# B&R Automation Studio project baseProject (part 2)

#### Main.st
```iecst
PROGRAM _INIT

	//Enable FBs and set parameters
	MpSequenceCore_0.Enable := TRUE;
	MpSequenceCore_0.Import := TRUE;
	MpSequenceCore_0.Mode := mpSEQUENCE_MODE_SINGLE_CYCLE;
	ParametersCore.Sequence := 'CoffeeSequence.xml';

	Timer.AxisLeft.PT := T#03s;
	Timer.AxisRight.PT := T#03s;
	Timer.Coffee.PT := T#03s;
	Timer.ExecuteWait.PT := T#03s;
	Timer.Start.PT := T#500ms;
	Timer.Stop.PT := T#01s;
	Timer.TakeOutCup.PT := T#01s;
	Timer.Wait.PT := T#03s;
	Timer.StopButton.PT := T#02s;
	Timer.CoffeeWait.PT := T#01s;

END_PROGRAM
PROGRAM _CYCLIC

	//Set FB parameters
	MpSequenceCore_0.MpLink := ADR(gSequenceCore);
	MpSequenceCore_0.Parameters := ADR(ParametersCore);

	IF MpSequenceCore_0.CommandDone AND MpSequenceCore_0.Import THEN
		MpSequenceCore_0.Import := FALSE;
	END_IF

	//Start if Start-Button is pressed
	IF SequenceStart AND MpSequenceCore_0.Info.ReadyToStart THEN
		MpSequenceCore_0.Start := TRUE;
		EditSequence := FALSE;
		MpSequenceCore_0.ErrorReset := FALSE;
	ELSE

		MpSequenceCore_0.Start := FALSE;
		CmdSeq.Start.MovementState := mpSEQUENCE_MOVEMENT_IDLE;
		CmdSeq.AxisLeft.MovementState := mpSEQUENCE_MOVEMENT_IDLE;
		CmdSeq.AxisRight.MovementState := mpSEQUENCE_MOVEMENT_IDLE;
		CmdSeq.Coffee.MovementState := mpSEQUENCE_MOVEMENT_IDLE;
		CmdSeq.End.MovementState := mpSEQUENCE_MOVEMENT_IDLE;
		CmdSeq.TakeOutCup.MovementState := mpSEQUENCE_MOVEMENT_IDLE;
		CmdSeq.Wait.MovementState := mpSEQUENCE_MOVEMENT_IDLE;
		Timer.AxisLeft.IN := FALSE;
		Timer.AxisRight.IN := FALSE;
		Timer.Coffee.IN := FALSE;
		Timer.ExecuteWait.IN := FALSE;
		Timer.Start.IN := FALSE;
		Timer.Stop.IN := FALSE;
		Timer.TakeOutCup.IN := FALSE;
		Timer.Wait.IN := FALSE;
		Timer.StopButton.IN := TRUE;

		Transform := '[{"select":"#g83","duration":1000,"translate":[3.497,-208.81101],"display":true}
		,{"select":"#rect999-9-2","duration":1000,"display":false}
		,{"select":"#rect999-1","duration":1000,"display":false}
		,{"select":"#path49","duration":2000,"fill":7}
		,{"select":"#path39","duration":2000,"fill":0}
		,{"select":"#path41","duration":2000,"fill":2}
		,{"select":"#path3","duration":2000,"fill":3}
		,{"select":"#gLamp1","duration":2000,"fill":7}
		,{"select":"#gLamp2","duration":2000,"fill":7}
		,{"select":"#gLamp3","duration":2000,"fill":7}
		,{"select":"#gLamp4","duration":2000,"fill":7}
		,{"select":"#gLamp5","duration":2000,"fill":7}
		,{"select":"#gLamp6","duration":2000,"fill":7}]';

		IF Timer.StopButton.Q THEN
			Timer.StopButton.IN := FALSE;
		END_IF

		EditSequence := TRUE;

	END_IF

	(****************************************************************START*********************************************************************)
	IF CmdSeq.Start.Start THEN

		CmdSeq.Start.MovementState := mpSEQUENCE_MOVEMENT_ACTIVE;
		Timer.Start.IN := TRUE;
		Transform := '[{"select":"#g83","duration":500,"display":true}]';
		IF Timer.Start.Q THEN
			Timer.Start.IN := FALSE;
			CmdSeq.Start.MovementState := mpSEQUENCE_MOVEMENT_DONE;
		END_IF

	ELSE
		CmdSeq.Start.MovementState := mpSEQUENCE_MOVEMENT_IDLE;
	END_IF

	(****************************************************************AXIS LEFT*********************************************************************)
	IF CmdSeq.AxisLeft.Start THEN

		CmdSeq.AxisLeft.MovementState := mpSEQUENCE_MOVEMENT_ACTIVE;
		Timer.AxisLeft.IN := TRUE;
		Transform := '[{"select":"#g83","duration":3000,"translate":[440,-208.81101]},{"select":"#gLamp1","duration":2000,"fill":8},{"select":"#gLamp4","duration":2000,"fill":8}]';
		IF Timer.AxisLeft.Q THEN
			Timer.AxisLeft.IN := FALSE;
			CmdSeq.AxisLeft.MovementState := mpSEQUENCE_MOVEMENT_DONE;
		END_IF
	ELSE
		CmdSeq.AxisLeft.MovementState := mpSEQUENCE_MOVEMENT_IDLE;
	END_IF

	(****************************************************************AXIS RIGHT*********************************************************************)
	IF CmdSeq.AxisRight.Start THEN

		CmdSeq.AxisRight.MovementState := mpSEQUENCE_MOVEMENT_ACTIVE;
		Timer.AxisRight.IN := TRUE;
		Transform := '[{"select":"#g83","duration":3000,"translate":[560,-208.81101]},{"select":"#gLamp3","duration":2000,"fill":10},{"select":"#gLamp6","duration":2000,"fill":10}]';
		IF Timer.AxisRight.Q THEN
			Timer.AxisRight.IN := FALSE;
			CmdSeq.AxisRight.MovementState := mpSEQUENCE_MOVEMENT_DONE;
		END_IF
	ELSE
		CmdSeq.AxisRight.MovementState := mpSEQUENCE_MOVEMENT_IDLE;
	END_IF

	(****************************************************************COFFEE*********************************************************************)
	IF CmdSeq.Coffee.Start THEN

		CmdSeq.Coffee.MovementState := mpSEQUENCE_MOVEMENT_ACTIVE;
		Timer.Coffee.IN := TRUE;
		Transform :='[{"select":"#path39","duration":2000,"fill":7}
		,{"select":"#path41","duration":2000,"fill":7}
		,{"select":"#path3","duration":2000,"fill":7}
		,{"select":"#gLamp2","duration":2000,"fill":9},
		{"select":"#gLamp5","duration":2000,"fill":9}]';
		IF Timer.Coffee.Q THEN

			Timer.ExecuteWait.IN := TRUE;

			Transform := '[{"select":"#rect999-9-2","duration":2000,"display":true,"fill":1}
			,{"select":"#rect999-1","duration":2000,"display":true,"fill":1}
			,{"select":"#path49","duration":2000,"fill":0}
			,{"select":"#path39","duration":2000,"fill":0}
			,{"select":"#path41","duration":2000,"fill":2}
			,{"select":"#path3","duration":2000,"fill":3}]';
			IF Timer.ExecuteWait.Q THEN

				Timer.CoffeeWait.IN := TRUE;
				Transform := '[{"select":"#rect999-1","duration":1000,"display":false},
				{"select":"#rect999-9-2","duration":1000,"display":false},
				{"select":"#path49","duration":1000,"fill":7}]';
				IF Timer.CoffeeWait.Q THEN
					Timer.CoffeeWait.IN := FALSE;
					Timer.Coffee.IN := FALSE;
					Timer.ExecuteWait.IN := FALSE;
					CmdSeq.Coffee.MovementState := mpSEQUENCE_MOVEMENT_DONE;
				END_IF
			END_IF
		END_IF

	ELSE
		CmdSeq.Coffee.MovementState := mpSEQUENCE_MOVEMENT_IDLE;
	END_IF

	(****************************************************************TAKEOUT*********************************************************************)
	IF CmdSeq.TakeOutCup.Start THEN

		CmdSeq.TakeOutCup.MovementState := mpSEQUENCE_MOVEMENT_ACTIVE;
		Timer.TakeOutCup.IN := TRUE;
		Transform := '[{"select":"#g83","duration":500,"display":false}]';
		IF Timer.TakeOutCup.Q THEN
			Timer.TakeOutCup.IN := FALSE;
			CmdSeq.TakeOutCup.MovementState := mpSEQUENCE_MOVEMENT_DONE;
		END_IF
	ELSE
		CmdSeq.TakeOutCup.MovementState := mpSEQUENCE_MOVEMENT_IDLE;
	END_IF

	(****************************************************************WAIT*********************************************************************)
	IF CmdSeq.Wait.Start THEN
		CmdSeq.Wait.MovementState := mpSEQUENCE_MOVEMENT_ACTIVE;
		Timer.Wait.IN := TRUE;

		IF Timer.Wait.Q THEN
			Timer.Wait.IN := FALSE;
			CmdSeq.Wait.MovementState := mpSEQUENCE_MOVEMENT_DONE;
		END_IF
	ELSE
		CmdSeq.Wait.MovementState := mpSEQUENCE_MOVEMENT_IDLE;
	END_IF

	(****************************************************************STOP*********************************************************************)
	IF CmdSeq.Stop.Start THEN
		CmdSeq.Stop.MovementState := mpSEQUENCE_MOVEMENT_ACTIVE;
		Timer.Stop.IN := TRUE;
		Transform := '[{"select":"#g83","duration":1000,"translate":[3.497,-208.81101]}
		]';

		IF Timer.Stop.Q THEN
			Timer.Stop.IN := FALSE;
			CmdSeq.Stop.MovementState := mpSEQUENCE_MOVEMENT_DONE;
			Transform := '[{"select":"#g83","duration":500,"display":true}]';
			SequenceStart := FALSE;
		END_IF
	ELSE
		CmdSeq.Stop.MovementState := mpSEQUENCE_MOVEMENT_IDLE;
	END_IF

	(****************************************************************ERROR*********************************************************************)
	IF MpSequenceCore_0.Error THEN
		SequenceStart := FALSE;
		MpSequenceCore_0.Import := FALSE;
		MpSequenceCore_0.ErrorReset := gCoffeeMainLogic.cmdClear;
	END_IF

	IF SavePressed THEN
		MpSequenceCore_0.Import := TRUE;
		SavePressed := FALSE;
	END_IF

	//Call FB
	MpSequenceCore_0();
	Timer.AxisLeft();
	Timer.AxisRight();
	Timer.Coffee();
	Timer.Start();
	Timer.Stop();
	Timer.TakeOutCup();
	Timer.Wait();
	Timer.ExecuteWait();
	Timer.StopButton();
	Timer.CoffeeWait();

END_PROGRAM
```

### Program Logical/Infrastructure/CodeBox (IEC) - CodeBox handling

#### Main.st
```iecst
PROGRAM _INIT

	State := WAIT;

END_PROGRAM

PROGRAM _CYCLIC

	//Set FB parameter
	MpCodeBoxCore_0(
	MpLink := ADR(gCodeBoxCore),
	Enable := TRUE,
	ErrorReset := gCoffeeMainLogic.cmdClear);

	CASE State OF
		WAIT:
			CodeBoxTransform := '[{"select":"#gLamp1","duration":200,"fill":7}
			,{"select":"#gLamp2","duration":200,"fill":7}
			,{"select":"#gLamp3","duration":200,"fill":7}
			,{"select":"#gLamp4","duration":200,"fill":7}
			,{"select":"#gLamp5","duration":200,"fill":7}
			,{"select":"#gLamp6","duration":200,"fill":7}]';

			IF gCoffeeMainLogic.PackMLState = 'Idle' THEN
				State := CUP_START_POS;

			END_IF

		CUP_START_POS:
			Cup.StartPosition := TRUE;
			IF Lamp.Green THEN

				CodeBoxTransform := '[{"select":"#gLamp1","duration":1000,"fill":10}
					,{"select":"#gLamp2","duration":1000,"fill":7}
					,{"select":"#gLamp3","duration":1000,"fill":7}
					,{"select":"#gLamp4","duration":1000,"fill":10}
					,{"select":"#gLamp5","duration":1000,"fill":7}
					,{"select":"#gLamp6","duration":1000,"fill":7}]';

			ELSIF Lamp.Red THEN
				CodeBoxTransform := '[{"select":"#gLamp1","duration":1000,"fill":8}
				,{"select":"#gLamp2","duration":1000,"fill":7}
				,{"select":"#gLamp3","duration":1000,"fill":7}
				,{"select":"#gLamp4","duration":1000,"fill":8}
				,{"select":"#gLamp5","duration":1000,"fill":7}
				,{"select":"#gLamp6","duration":1000,"fill":7}]';

			ELSIF Lamp.Yellow THEN
				CodeBoxTransform := '[{"select":"#gLamp1","duration":1000,"fill":9}
				,{"select":"#gLamp2","duration":1000,"fill":7}
				,{"select":"#gLamp3","duration":1000,"fill":7}
				,{"select":"#gLamp4","duration":1000,"fill":9}
				,{"select":"#gLamp5","duration":1000,"fill":7}
				,{"select":"#gLamp6","duration":1000,"fill":7}]';
			ELSE
				CodeBoxTransform := '[{"select":"#gLamp1","duration":1000,"fill":7}
				,{"select":"#gLamp2","duration":1000,"fill":7}
				,{"select":"#gLamp3","duration":1000,"fill":7}
				,{"select":"#gLamp4","duration":1000,"fill":7}
				,{"select":"#gLamp5","duration":1000,"fill":7}
				,{"select":"#gLamp6","duration":1000,"fill":7}]';
			END_IF

			IF gCoffeeMainLogic.PackMLState = 'Execute' THEN
				State := CUP_COFFEE;
				Cup.StartPosition := FALSE;
			END_IF

		CUP_COFFEE:
			Cup.CoffeePosition := TRUE;
			IF gCoffeeMainLogic.PackMLState = 'Completing' THEN
				State := CUP_END_POS;
				Cup.CoffeePosition := FALSE;
			END_IF

			IF Lamp.Green THEN

				CodeBoxTransform := '[{"select":"#gLamp1","duration":1000,"fill":7}
				,{"select":"#gLamp2","duration":1000,"fill":10}
				,{"select":"#gLamp3","duration":1000,"fill":7}
				,{"select":"#gLamp4","duration":1000,"fill":7}
				,{"select":"#gLamp5","duration":1000,"fill":10}
				,{"select":"#gLamp6","duration":1000,"fill":7}]';

			ELSIF Lamp.Red THEN
				CodeBoxTransform := '[{"select":"#gLamp1","duration":1000,"fill":7}
				,{"select":"#gLamp2","duration":1000,"fill":8}
				,{"select":"#gLamp3","duration":1000,"fill":7}
				,{"select":"#gLamp4","duration":1000,"fill":7}
				,{"select":"#gLamp5","duration":1000,"fill":8}
				,{"select":"#gLamp6","duration":1000,"fill":7}]';

			ELSIF Lamp.Yellow THEN
				CodeBoxTransform := '[{"select":"#gLamp1","duration":1000,"fill":7}
				,{"select":"#gLamp2","duration":1000,"fill":9}
				,{"select":"#gLamp3","duration":1000,"fill":7}
				,{"select":"#gLamp4","duration":1000,"fill":7}
				,{"select":"#gLamp5","duration":1000,"fill":9}
				,{"select":"#gLamp6","duration":1000,"fill":7}]';
			ELSE
				CodeBoxTransform := '[{"select":"#gLamp1","duration":1000,"fill":7}
				,{"select":"#gLamp2","duration":1000,"fill":7}
				,{"select":"#gLamp3","duration":1000,"fill":7}
				,{"select":"#gLamp4","duration":1000,"fill":7}
				,{"select":"#gLamp5","duration":1000,"fill":7}
				,{"select":"#gLamp6","duration":1000,"fill":7}]';
			END_IF
		CUP_END_POS:
			Cup.EndPosition := TRUE;
			IF Lamp.Green THEN

				CodeBoxTransform := '[{"select":"#gLamp1","duration":1000,"fill":7}
				,{"select":"#gLamp2","duration":1000,"fill":7}
				,{"select":"#gLamp3","duration":1000,"fill":10}
				,{"select":"#gLamp4","duration":1000,"fill":7}
				,{"select":"#gLamp5","duration":1000,"fill":7}
				,{"select":"#gLamp6","duration":1000,"fill":10}]';

			ELSIF Lamp.Red THEN
				CodeBoxTransform := '[{"select":"#gLamp1","duration":1000,"fill":7}
				,{"select":"#gLamp2","duration":1000,"fill":7}
				,{"select":"#gLamp3","duration":1000,"fill":8}
				,{"select":"#gLamp4","duration":1000,"fill":7}
				,{"select":"#gLamp5","duration":1000,"fill":7}
				,{"select":"#gLamp6","duration":1000,"fill":8}]';

			ELSIF Lamp.Yellow THEN
				CodeBoxTransform := '[{"select":"#gLamp1","duration":1000,"fill":7}
				,{"select":"#gLamp2","duration":1000,"fill":7}
				,{"select":"#gLamp3","duration":1000,"fill":9}
				,{"select":"#gLamp4","duration":1000,"fill":7}
				,{"select":"#gLamp5","duration":1000,"fill":7}
				,{"select":"#gLamp6","duration":1000,"fill":9}]';
			ELSE
				CodeBoxTransform := '[{"select":"#gLamp1","duration":1000,"fill":7}
				,{"select":"#gLamp2","duration":1000,"fill":7}
				,{"select":"#gLamp3","duration":1000,"fill":7}
				,{"select":"#gLamp4","duration":1000,"fill":7}
				,{"select":"#gLamp5","duration":1000,"fill":7}
				,{"select":"#gLamp6","duration":1000,"fill":7}]';
			END_IF
			IF gCoffeeMainLogic.PackMLState = 'Idle' THEN
				State := WAIT;
				Cup.EndPosition := FALSE;
			END_IF

	END_CASE

END_PROGRAM
```

### Program Logical/Infrastructure/Skyline (IEC)

#### Types.typ
```iecst
TYPE
	Module_Type : 	STRUCT
		Notification : ARRAY[0..7]OF STRING[80] := [8('Information: Module ok!')];
		Name : ARRAY[0..7]OF STRING[50] := ['Start','Water_Tank','Coffee_Tank','Milk_Tank','Filtering','Sugar_Tank','Coffee_Grinder','End'];
		IngredientLevel : ARRAY[0..7]OF INT := [8(1000)];
		AlarmFlag : ARRAY[0..7]OF BOOL;
		AlarmName : ARRAY[0..7]OF STRING[80] := ['','WaterEmpty','CoffeeEmpty','MilkEmpty','','SugarEmpty',2('')];
		Option : Option_Type;
		ShowOption : BOOL;
		AcknowledgeFlag : ARRAY[0..7]OF BOOL := [8(TRUE)];
	END_STRUCT;
	SkylineStateEnum :
		(
		WAIT,
		ACTIVATE,
		DEACTIVATE,
		NOTIFICATION,
		DEACTIVATE_NOTIFICATION,
		ACTIVATE_OPTION,
		DEACTIVATE_OPTION
		);
	SkylineCmd_Type : 	STRUCT
		Activate : BOOL;
		Deactivate : BOOL;
		Notification : BOOL;
		DeactivateOption : BOOL;
		ActivateOption : BOOL;
	END_STRUCT;
	Option_Type : 	STRUCT
		StateOFF : ARRAY[0..3]OF STRING[80] := [2('Off'),'NormalFilter','GrindRough'];
		StateON : ARRAY[0..3]OF STRING[80] := ['Cooling','Heating','PremiumFilter','GrindFine'];
		Name : ARRAY[0..3]OF STRING[80] := ['OptionCooling','OptionHeating','OptionFilter','OptionGrinder'];
		Activate : ARRAY[0..3]OF INT;
		Modules : ARRAY[0..3]OF STRING[80] := [2('Water_Tank'),'Filtering','Coffee_Grinder'];
	END_STRUCT;
END_TYPE
```

#### Variables.var
```iecst
VAR CONSTANT
	LEVEL_LIMIT : USINT := 250;
	ON : INT := 1;
	ACTIVATION : INT := 50;
	MAX_MODULES : USINT := 7;
	MAX_OPTIONS : USINT := 3;
END_VAR
VAR
	x : INT := 0;
	y : USINT := 0;
	i : USINT := 0;
	Cmd : SkylineCmd_Type := (0);
	Step : SkylineStateEnum := WAIT;
	Module : Module_Type;
	BlockDeactivate : BOOL := TRUE;
	State : STRING[50] := 'Off';
	BlockActivate : BOOL := TRUE;
	SelectedModuleIndex : INT := 0;
	BlockFunctions : BOOL := FALSE;
	Active : BOOL := 0;
	SkylineNotification : STRING[80] := '';
	Deactive : BOOL := TRUE;
	z : INT := 0;
END_VAR
```

#### Main.st
```iecst
PROGRAM _CYCLIC

	//Get ingredient level
	Module.IngredientLevel[1] := gCoffeeMainLogic.AlarmRefill[3];
	Module.IngredientLevel[2] := gCoffeeMainLogic.AlarmRefill[0];
	Module.IngredientLevel[3] := gCoffeeMainLogic.AlarmRefill[1];
	Module.IngredientLevel[5] := gCoffeeMainLogic.AlarmRefill[2];

	SkylineNotification := Module.Notification[SelectedModuleIndex];

	//Check if ingredient got 0
	FOR x := 0 TO MAX_MODULES DO
		IF Module.IngredientLevel[x] = 0 THEN
			Module.AlarmFlag[x] := TRUE;
			Module.AcknowledgeFlag[x] := FALSE;
		ELSE
			Module.AlarmFlag[x] := FALSE;
		END_IF
	END_FOR

	CASE Step OF
		WAIT:

			IF Cmd.Activate THEN
				Step := ACTIVATE;
				BlockDeactivate := FALSE;
				BlockFunctions := FALSE;
				State := 'Ready';

			ELSIF Cmd.Deactivate THEN
				Step := DEACTIVATE;
				BlockActivate := FALSE;
				BlockFunctions := FALSE;
				Active := FALSE;
				State := 'Off';

			ELSIF Cmd.ActivateOption THEN
				Step := ACTIVATE_OPTION;
				Cmd.ActivateOption := FALSE;

			ELSIF Cmd.DeactivateOption THEN
				Step := DEACTIVATE_OPTION;
				Cmd.DeactivateOption := FALSE;
			END_IF

			IF i > MAX_MODULES THEN
				i := 0;
			END_IF

		ACTIVATE:

			Active := TRUE;
			Deactive := FALSE;

			IF y <= ACTIVATION THEN

				y := y + 1;

				IF i <= MAX_MODULES AND y = ACTIVATION THEN

					//Check module state
					IF Module.AlarmFlag[i] OR Module.AcknowledgeFlag[i] = FALSE THEN
						MpSkylineSetModuleState(gSkyline, Module.Name[i], 'Error');
					ELSE

						MpSkylineSetModuleState(gSkyline, Module.Name[i], 'Ready');
					END_IF

					//Check notification
					IF Module.IngredientLevel[i] <= LEVEL_LIMIT THEN
						MpSkylineSetNotification(gSkyline, Module.Name[i], 'Information');
						Module.Notification[i] := 'Information: Module ok!';
					END_IF

					//Check alarm
					IF Module.AcknowledgeFlag[i] = FALSE THEN
						MpSkylineSetNotification(gSkyline, Module.Name[i], 'Alarm');
					END_IF

					i := i + 1;
					y := 0;

				ELSIF i > MAX_MODULES THEN
					Step := WAIT;
					BlockDeactivate := TRUE;
					BlockFunctions := TRUE;
					Cmd.Activate := FALSE;
				END_IF
			END_IF

		DEACTIVATE:

			IF y <= ACTIVATION THEN

				y := y + 1;

				IF i <= MAX_MODULES AND y = ACTIVATION THEN
					MpSkylineSetModuleState(gSkyline, Module.Name[i], 'Off');
					MpSkylineResetNotification(gSkyline, Module.Name[i], 'Alarm');
					MpSkylineResetNotification(gSkyline, Module.Name[i], 'Information');
					i := i + 1;
					y := 0;

				ELSIF i > MAX_MODULES THEN
					Step := WAIT;
					BlockActivate := TRUE;
					Cmd.Deactivate := FALSE;
					Deactive := TRUE;
				END_IF
			END_IF

		ACTIVATE_OPTION:

			Module.ShowOption := TRUE;

			FOR i := 0 TO MAX_OPTIONS DO

				IF Module.Option.Activate[i] = ON THEN
					MpSkylineSetOptionState(gSkyline, Module.Option.Modules[i], Module.Option.Name[i], Module.Option.StateON[i]);
				ELSE
					MpSkylineSetOptionState(gSkyline, Module.Option.Modules[i], Module.Option.Name[i], Module.Option.StateOFF[i]);
				END_IF

			END_FOR;

			Step := WAIT;
			i := 0;

		DEACTIVATE_OPTION:

			Module.ShowOption := FALSE;
			Step := WAIT;

	END_CASE

	//Check notification an status
	IF BlockFunctions  THEN

		FOR z := 0 TO MAX_MODULES DO
			// Set and reset information
			IF Module.IngredientLevel[z] <= LEVEL_LIMIT THEN
				MpSkylineSetNotification(gSkyline, Module.Name[z], 'Information');
				Module.Notification[z] := 'Information: Fill level below limit!';
			ELSE
				MpSkylineResetNotification(gSkyline, Module.Name[z], 'Information');
				Module.Notification[z] := 'Information: Module ok!';
			END_IF

			//Set alarm
			IF Module.AlarmFlag[z] THEN
				MpSkylineSetNotification(gSkyline, Module.Name[z], 'Alarm');
				MpSkylineSetModuleState(gSkyline, Module.Name[z], 'Error');
				Module.Notification[z] := 'Alarm: Fill level too low!';

				//Reset alarm
			ELSIF MpAlarmXCheckState(gAlarmXCore, Module.AlarmName[z], mpALARMX_STATE_NONE) AND Module.AcknowledgeFlag[z] = FALSE THEN
				MpSkylineResetNotification(gSkyline, Module.Name[z], 'Alarm');
				MpSkylineSetModuleState(gSkyline, Module.Name[z], State);
				Module.AcknowledgeFlag[z] := TRUE;

				//Check ingredients level
				IF Module.IngredientLevel[z] <= LEVEL_LIMIT THEN
					Module.Notification[z] := 'Information: Fill level below limit!';
					MpSkylineSetNotification(gSkyline, Module.Name[z], 'Information');
				ELSE
					Module.Notification[z] := 'Information: Module ok!';
					MpSkylineSetNotification(gSkyline, Module.Name[z], 'Information');
				END_IF
			END_IF
		END_FOR

		z := 0;

	END_IF

END_PROGRAM
```

### Package Logical/Industry - Industry Components

### Program Logical/Industry/PackML (IEC) - PackML handling

#### Variables.var
```iecst
VAR
	MpPackMLBasicUI_0 : MpPackMLBasicUI; (*MpPackMLBasicUI instance*)
	MpPackMLBasicUIConnect : MpPackMLBasicUIConnectType := (ModeControl:=(SelectedIndex:=1)); (*MpPackMLBasicUI UI connection datapoints*)
	MpPackMLStatisticsUI_0 : MpPackMLStatisticsUI; (*MpPackMLStatisticsUI instance*)
	MpPackMLStatisticsUIConnect : MpPackMLStatisticsUIConnectType; (*MpPackMLStatistics UI connection datapoints*)
	MpPackMLMode_0 : MpPackMLMode;
	MpPackMLMode_1 : MpPackMLMode;
END_VAR
```

#### Main.st
```iecst
PROGRAM _INIT

END_PROGRAM

PROGRAM _CYCLIC

	//Set FB parameters

	MpPackMLMode_0(
		MpLink := ADR(gPackMLStandaloneUnit),
		Enable := TRUE,
		ModeID := PACKML_MODE_PRODUCTION,
		Start := gCoffeeMainLogic.cmdStart,
		Stop := gCoffeeMainLogic.cmdStop,
		Reset := MpPackMLStateIsActive(gPackMLStandaloneUnit,mpPACKML_STATE_STOPPED,PACKML_MODE_PRODUCTION),
		Abort := (gCoffeeMainLogic.cmdAbort AND MpPackMLMode_0.ModeActive),
		Clear := gCoffeeMainLogic.cmdClear);

	MpPackMLMode_1(
		MpLink := ADR(gPackMLStandaloneUnit),
		Enable := TRUE,
		ModeID := PACKML_MODE_MAINTENANCE);

	MpPackMLBasicUI_0(
		MpLink := ADR(gPackMLStandaloneUnit),
		Enable := TRUE,
		UIConnect := ADR(MpPackMLBasicUIConnect));

	MpPackMLStatisticsUI_0(
		MpLink := ADR(gPackMLStandaloneUnit),
		Enable := TRUE,
		UIConnect := ADR(MpPackMLStatisticsUIConnect));

	//Check if you can refill the ingredients
	IF MpPackMLBasicUIConnect.StateCurrent = mpPACKML_STATE_IDLE OR MpPackMLBasicUIConnect.StateCurrent = mpPACKML_STATE_ABORTED THEN
		gCoffeeMainLogic.IdleState := TRUE;
	ELSE
		gCoffeeMainLogic.IdleState := FALSE;
	END_IF

END_PROGRAM
```

### Program Logical/MainControl (IEC) - MainContol program

#### Cyclic.st - Cyclic code
```iecst
PROGRAM _CYCLIC

	// Main state machine for the brewing process handled by PackML
(****************************************************************IDLE*********************************************************************)

	IF (MpPackMLStateIsActive(gPackMLStandaloneUnit, mpPACKML_STATE_IDLE, PACKML_MODE_PRODUCTION)) THEN
		gCoffeeMainLogic.PackMLState := 'Idle';
		TransitionTime := 500;
		TransformTime := T#500ms;
		gCoffeeMainLogic.AxisCupFeeder.Power 		:= TRUE;
		gCoffeeMainLogic.AxisTakeout.Power 			:= TRUE;

		IF (gCoffeeMainLogic.AxisTakeout.Active = TRUE) AND (gCoffeeMainLogic.AxisCupFeeder.Active = TRUE)  THEN

			Transform := '[{"select":"#g83","duration":500,"display":true}]';
		ELSE

			gCoffeeMainLogic.cmdAbort := TRUE;

		END_IF

	END_IF

	(****************************************************************RESETTING*********************************************************************)

	IF (MpPackMLStateIsActive(gPackMLStandaloneUnit, mpPACKML_STATE_RESETTING
		, PACKML_MODE_PRODUCTION)) THEN
		gCoffeeMainLogic.PackMLState := 'Resetting';
		gCoffeeMainLogic.cmdClear 		:= FALSE;
		gCoffeeMainLogic.cmdAbort 		:= FALSE;

		gCoffeeMainLogic.AxisCupFeeder.Power 		:= TRUE;				// power and home both conveyor axes
		gCoffeeMainLogic.AxisTakeout.Power 			:= TRUE;

		IF(gCoffeeMainLogic.AxisTakeout.PowerOn = TRUE) AND (gCoffeeMainLogic.AxisCupFeeder.PowerOn = TRUE)  THEN

			MpPackMLStateComplete(gPackMLStandaloneUnit, PACKML_MODE_PRODUCTION);

		END_IF
	END_IF

	(******************************************************************STARTING*******************************************************************)

	IF (MpPackMLStateIsActive(gPackMLStandaloneUnit, mpPACKML_STATE_STARTING, PACKML_MODE_PRODUCTION)) THEN
		gCoffeeMainLogic.PackMLState := 'Starting';
		TransitionTime := 3000;
		Transform := '[{"select":"#g83","duration":3000,"translate":[375,-87.299533]}]';
		TransformTime := T#3S;
		TransformWait.IN := TRUE;
		TransformWait.PT := TransformTime;

		gCoffeeMainLogic.AxisCupFeeder.MoveAdditive 	:= TRUE;			// start moving the cup to fill station
		gCoffeeMainLogic.cmdStart := FALSE;

		IF (gCoffeeMainLogic.AxisCupFeeder.InPosition) AND TransformWait.Q = TRUE THEN
			TransformWait.IN := FALSE;
			gCoffeeMainLogic.AxisCupFeeder.MoveAdditive 	:= FALSE;				// reset command when in position
			gCoffeeMainLogic.AxisCupFeeder.InPosition := FALSE;
			gCoffeeMainLogic.AxisCupFeeder.Position 	:= 0.0;
			MpPackMLStateComplete(gPackMLStandaloneUnit, PACKML_MODE_PRODUCTION);
			TransformWait();
		END_IF

	END_IF

	(******************************************************************EXECUTE*******************************************************************)

	IF (MpPackMLStateIsActive(gPackMLStandaloneUnit, mpPACKML_STATE_EXECUTE, PACKML_MODE_PRODUCTION)) THEN
		gCoffeeMainLogic.PackMLState := 'Execute';
		TransitionTime := 3000;
		TransformTime := T#3S;
		Transform :='[{"select":"#path39","duration":2000,"fill":7}
		,{"select":"#path41","duration":2000,"fill":7}
		,{"select":"#path3","duration":2000,"fill":7}
		,{"select":"#rect999","duration":2000,"display":true,"fill":1}
		,{"select":"#rect999-9","duration":2000,"display":true,"fill":1}
		,{"select":"#path49","duration":2000,"fill":0}]';
		ExecuteWait.IN := TRUE;
		ExecuteWait.PT := TransformTime;
		ExecuteWait();

		IF ExecuteWait.Q = TRUE THEN
			FillCoffeeWait.IN := TRUE;
			FillCoffeeWait.PT := T#2s;
			Transform := '[{"select":"#path49","duration":2000,"fill":0}
			,{"select":"#path39","duration":2000,"fill":0}
			,{"select":"#path41","duration":2000,"fill":2}
			,{"select":"#path3","duration":2000,"fill":3}
			,{"select":"#rect999","duration":500,"display":false}
			,{"select":"#rect999-9","duration":500,"display":false}
			,{"select":"#path49","duration":2000,"fill":7}]';

			IF FillCoffeeWait.Q THEN
				FillCoffeeWait.IN := FALSE;
				ExecuteWait.IN := FALSE;
				gCoffeeMainLogic.AxisTakeout.MoveAdditive := TRUE;					// start moving cup to take out
				MpPackMLStateComplete(gPackMLStandaloneUnit, PACKML_MODE_PRODUCTION);
			END_IF
		END_IF

	END_IF

	(******************************************************************Completing*******************************************************************)

	IF (MpPackMLStateIsActive(gPackMLStandaloneUnit, mpPACKML_STATE_COMPLETING, PACKML_MODE_PRODUCTION)) THEN
		TransitionTime := 3000;
		Transform := '[{"select":"#g83","duration":3000,"translate":[560,-87.299533]}]';
		gCoffeeMainLogic.PackMLState := 'Completing';
		TransformWait.IN := TRUE;
		TransformWait.PT := TransformTime;

		IF (gCoffeeMainLogic.AxisTakeout.InPosition) AND TransformWait.Q = TRUE THEN

			TransitionTime := 500;
			Transform := '[{"select":"#g83","duration":500,"display":false}]';
			TransformHide.IN := TRUE;
			TransformHide.PT := TransformTime;

			IF TransformHide.Q = TRUE THEN

				CupHideWait.IN := TRUE;
				CupHideWait.PT := T#1S;
				Transform := '[{"select":"#g83","duration":1000,"translate":[3.497,-87.299533]}]';

				IF CupHideWait.Q = TRUE THEN
					CupHideWait.IN := FALSE;
					TransformWait.IN := FALSE;
					TransformHide.IN := FALSE;
					gCoffeeMainLogic.cmdStart					:= FALSE;					// reset the brewing start command
					gCoffeeMainLogic.AxisTakeout.MoveAdditive 	:= FALSE;					// reset command when in position
					gCoffeeMainLogic.AxisTakeout.InPosition := FALSE;
					gCoffeeMainLogic.AxisTakeout.Position 	:= 0.0;
					MpPackMLStateComplete(gPackMLStandaloneUnit, PACKML_MODE_PRODUCTION);
				END_IF

			END_IF

		END_IF

	END_IF
	TransformWait();
	CupHideWait();
	TransformHide();
	(****************************************************************STOPPED*********************************************************************)

	IF (MpPackMLStateIsActive(gPackMLStandaloneUnit, mpPACKML_STATE_STOPPED, PACKML_MODE_PRODUCTION)) THEN
		gCoffeeMainLogic.PackMLState := 'Stopped';
		gCoffeeMainLogic.cmdClear := FALSE;

	END_IF

	(******************************************************************ABORTING*******************************************************************)

	IF (MpPackMLStateIsActive(gPackMLStandaloneUnit, mpPACKML_STATE_ABORTING, PACKML_MODE_PRODUCTION)) THEN
		gCoffeeMainLogic.PackMLState := 'Aborting';
		gCoffeeMainLogic.AxisCupFeeder.Power 	:= FALSE;
		gCoffeeMainLogic.AxisTakeout.Power 		:= FALSE;

		IF (gCoffeeMainLogic.AxisCupFeeder.PowerOn = FALSE) AND (gCoffeeMainLogic.AxisTakeout.PowerOn = FALSE) THEN
			MpPackMLStateComplete(gPackMLStandaloneUnit, PACKML_MODE_PRODUCTION);
		END_IF

		gCoffeeMainLogic.cmdAbort := FALSE;
	END_IF

	(******************************************************************ABORTED*******************************************************************)

	IF (MpPackMLStateIsActive(gPackMLStandaloneUnit, mpPACKML_STATE_ABORTED, PACKML_MODE_PRODUCTION)) THEN
		gCoffeeMainLogic.PackMLState := 'Aborted';
		gCoffeeMainLogic.AxisCupFeeder.Power 			:= FALSE;
		gCoffeeMainLogic.AxisTakeout.Power 				:= FALSE;
		gCoffeeMainLogic.AxisCupFeeder.MoveAdditive 	:= FALSE;
		gCoffeeMainLogic.AxisTakeout.MoveAdditive		:= FALSE;
		gCoffeeMainLogic.AxisCupFeeder.Home			 	:= FALSE;
		gCoffeeMainLogic.AxisTakeout.Home				:= FALSE;
		gCoffeeMainLogic.cmdStart						:= FALSE;

		IF (gCoffeeMainLogic.AxisCupFeeder.PowerOn = FALSE) AND (gCoffeeMainLogic.AxisTakeout.PowerOn = FALSE) THEN
			MpPackMLStateComplete(gPackMLStandaloneUnit, PACKML_MODE_PRODUCTION);
		END_IF

		gCoffeeMainLogic.cmdAbort := FALSE;
	END_IF

	(******************************************************************END OF PACKML*******************************************************************)

	//Check if Alarm can be cleared
	IF (gClearAlarm = TRUE) THEN
		MainCoffeeUIConnect.visShowClearButton := YES;
	ELSE
		MainCoffeeUIConnect.visShowClearButton := NO;
	END_IF

	//Control Refill Alarms
	IF MainCoffeeUIConnect.visStartCoffee = TRUE THEN
		gCoffeeMainLogic.cmdStart := TRUE;
		(*gCoffeeMainLogic.cmdClear := TRUE*)
		MainCoffeeUIConnect.visStartCoffee := FALSE;
		ProducedCoffee.Number := ProducedCoffee.Number + 1;

		FOR i := 0 TO MAX_INGREDIENTS DO

			Refill[i] := Refill[i] - gCoffeeMainLogic.Refill[i];

			IF(Refill[i] < 0 ) THEN
				Refill[i] := 0;
			END_IF
		END_FOR;
	END_IF

	FOR i := 0 TO MAX_INGREDIENTS DO
		gCoffeeMainLogic.AlarmRefill[i] := Refill[i];
	END_FOR

	//Get correct measurement system
	IF gUnit = 'metric' THEN

		gSetUnit := 1;

	ELSIF gUnit = 'imperial' THEN
		gSetUnit := 2;

	ELSE
		gSetUnit := 3;

	END_IF;

	TransformWait();
	FillCoffeeWait();
	ExecuteWait();

END_PROGRAM
```

#### Variables.var - Local variables
```iecst
VAR
	FillCoffeeWait : TON := (0);
	ProducedCoffee : ProducedCoffeeType := (0);
	MainCoffeeUIConnect : MainCoffeeUIConnectType; (*Control structure of main logic*)
END_VAR
VAR CONSTANT
	YES : BOOL := FALSE; (*Display an element on the visualization screen*)
	NO : BOOL := TRUE; (*Hide an element on the visualization screen*)
END_VAR
VAR
	i : INT := 0;
END_VAR
VAR CONSTANT
	MAX_INGREDIENTS : INT := 3;
END_VAR
VAR
	Refill : ARRAY[0..3] OF INT := [4(500)];
	Transform : STRING[1000000] := ''; (*transforms the svg image in the coffee Visualization*)
	TransformTime : TIME := T#3S;
	TransformWait : TON := (0);
	TransitionTime : UINT := 3000;
	ExecuteWait : TON;
	CupHideWait : TON := (0);
	TransformHide : TON;
END_VAR
```

#### Types.typ - Local types
```iecst
TYPE
	ProducedCoffeeType : 	STRUCT
		Number : INT;
		_Number : INT;
		Name : STRING[80];
	END_STRUCT;
	RefillMainType : 	STRUCT
		Milk : INT; (*Whole amount of milk*)
		Sugar : INT; (*Whole amount of sugar*)
		Coffee : INT; (*Whole amount of coffee*)
		Water : INT; (*Whole amount of water*)
	END_STRUCT;
	RecipeSelectEnum :
		( (*Enumeration definition for recipe selection*)
		MAPP_REGULAR := 0,
		MAPP_MILKCOFFEE := 1,
		MAPP_ESSPRESSO := 2,
		MAPP_CAPPUCINO := 3,
		NO_SELECTION := 4
		);
	MainControlStepEnum :
		( (*Enumeration definition for main state machine*)
		STATE_IDLE,
		STATE_STARTING,
		STATE_EXECUTE,
		STATE_COMPLETING,
		STATE_TAKEOUT_CUP,
		STATE_POSITION_CUP
		);
	RefillStateEnum :
		( (*Enumeration definition for refill machine*)
		REFILL_NONE := 1,
		REFILL_WATER := 2,
		REFILL_MILK := 3,
		REFILL_COFFEE := 4,
		REFILL_SUGAR := 5
		);
	MainCoffeeUIConnectType : 	STRUCT  (*Main logic structure *)
		visShowClearButton : BOOL; (*HMI control bit*)
		visStartCoffee : BOOL; (*HMI control bit*)
	END_STRUCT;
END_TYPE
```

### Program Logical/ConveyorSim (IEC) - Conveyor simulation

#### Cyclic.st - Cyclic code
```iecst
PROGRAM _CYCLIC
//	Cupfeed conveyor simulation
	IF (gCoffeeMainLogic.AxisCupFeeder.Active = TRUE)   THEN
		IF (gCoffeeMainLogic.AxisCupFeeder.Power = TRUE) THEN
			gCoffeeMainLogic.AxisCupFeeder.PowerOn 	:= TRUE;
			ActivePowerCupFeeder := 30;
			IF (gCoffeeMainLogic.AxisCupFeeder.MoveAdditive = TRUE) THEN
				IF (gCoffeeMainLogic.AxisCupFeeder.Position < 700.0) THEN
					gCoffeeMainLogic.AxisCupFeeder.Position 	:=
					gCoffeeMainLogic.AxisCupFeeder.Position + 1.5;
					ActivePowerCupFeeder := 80;
				ELSE
					gCoffeeMainLogic.AxisCupFeeder.InPosition := TRUE;

					ActivePowerCupFeeder := 30;
				END_IF;
			END_IF;
		ELSE
			gCoffeeMainLogic.AxisCupFeeder.PowerOn 	:= FALSE;
			ActivePowerCupFeeder := 0;
		END_IF;
	ELSE
		gCoffeeMainLogic.AxisCupFeeder.PowerOn 	:= FALSE;

		ActivePowerCupFeeder := 0;
	END_IF;

	//	Takeout conveyor simulation
	IF (gCoffeeMainLogic.AxisTakeout.Active = TRUE)   THEN
		IF (gCoffeeMainLogic.AxisTakeout.Power = TRUE) THEN
			gCoffeeMainLogic.AxisTakeout.PowerOn 	:= TRUE;
			ActivePowerTakeout := 10;
			IF (gCoffeeMainLogic.AxisTakeout.MoveAdditive = TRUE) THEN
				IF (gCoffeeMainLogic.AxisTakeout.Position < 300.0) THEN
					gCoffeeMainLogic.AxisTakeout.Position 	:=
					gCoffeeMainLogic.AxisTakeout.Position + 1.5;
					ActivePowerTakeout := 68;
				ELSE
					gCoffeeMainLogic.AxisTakeout.InPosition := TRUE;

					ActivePowerTakeout := 10;
				END_IF;
			END_IF;
		ELSE
			gCoffeeMainLogic.AxisTakeout.PowerOn 	:= FALSE;
			ActivePowerTakeout := 0;
		END_IF;
	ELSE
		gCoffeeMainLogic.AxisTakeout.PowerOn 	:= FALSE;

		ActivePowerTakeout := 0;
	END_IF;

END_PROGRAM
```

#### Variables.var
```iecst
VAR
	ActivePowerCupFeeder : INT := 0;
	ActivePowerTakeout : INT := 0;
END_VAR
```

Listed in the project but not available here: Logical/motion, Logical/Documentation, Logical/ConveyorSim/Init.st, Logical/UserFiles
